{attribute 'GeneratedUsingTerminal: EL2014-0000-0016'}
{attribute addProperty BoxType "EL2014-0000-0016"}
{attribute addProperty Id "Channel_1AT %I*Channel_EA8D33D74Channel_2AT %I*Channel_EA8D33D74Channel_3AT %I*Channel_EA8D33D74Channel_4AT %I*Channel_EA8D33D74"}
{attribute addProperty CRC "1492378280"}
{attribute addProperty Size "16"}
TYPE DIG_Diag_Inputs_58F3E2A8 :
STRUCT
	{attribute addProperty Name "Channel_1"}
	Channel_1 AT %I* : Channel_EA8D33D7;
	{attribute addProperty Name "Channel_2"}
	Channel_2 AT %I* : Channel_EA8D33D7;
	{attribute addProperty Name "Channel_3"}
	Channel_3 AT %I* : Channel_EA8D33D7;
	{attribute addProperty Name "Channel_4"}
	Channel_4 AT %I* : Channel_EA8D33D7;
END_STRUCT
END_TYPE

(* stored: Version 1.2.0.0, ProductVersion 3.1.4024.9
   DUT DIG_Diag_Inputs_58F3E2A8: Id {aab2a7a0-6bb1-435a-aa3f-e3febf96020b} *)
